TYPE E_DecisionState :
(
	none := 0,
	Wait := 1,
	WayToJunction := 2,
	OnJunction := 3,
	Processed := 4,
	DriveOut := 5,
	Finished := 6,
	MAX_E_DecisionState
);
END_TYPE

(* stored: Version 1.1.0.1, ProductVersion 3.1.0.23
   DUT E_DecisionState: Id {7266c7fa-7dd8-476c-90b1-afa9d4adfbc2} *)
